FUNCTION_BLOCK FB_methods
VAR_INPUT
END_VAR
VAR_OUTPUT
	StartIntegration : BOOL;
END_VAR
VAR
END_VAR


IF StartIntegration THEN
	FIFOaxis.M_Integrate();
	StartIntegration := FALSE;
END_IF

{attribute 'TcRpcEnable'}
METHOD M_Integrate : BOOL
VAR_INPUT
END_VAR

StartIntegration := TRUE;
END_METHOD

END_FUNCTION_BLOCK

(* stored: Version 1.1.0.1, ProductVersion 3.1.4024.9
   POU FB_methods: Id {97d15662-671b-4aec-b908-838048d1d643}, SpecialFunc None
   Method M_Integrate: Id {d58f5ba4-03c5-4fb1-8281-0bc58fcc5113} *)
